// TIA Portal V16 export
// export: Created 2024-04-15T10:45:14.7081519Z, ExportSetting WithDefaults, DisplayName Totally Integrated Automation Portal, DisplayVersion V16 Update 6, DisplayName TIA Portal Version Control Interface, DisplayVersion V16 Update 2, DisplayName TIA Portal Openness, DisplayVersion V16 Update 6, DisplayName TIA Portal Test Suite Advanced, DisplayVersion V16, DisplayName SINAMICS Startdrive Advanced, DisplayVersion V16 Update 5, DisplayName SINAMICS Startdrive G130, G150, S120, S150, SINAMICS MV, S210, DisplayVersion V16 Update 5, DisplayName SINAMICS Startdrive G110M, G120, G120C, G120D, G120P, G115D, DisplayVersion V16 Update 5, DisplayName STEP 7 Professional, DisplayVersion V16 Update 6, DisplayName STEP 7 Safety, DisplayVersion V16, DisplayName WinCC Advanced, DisplayVersion V16 Update 6
FUNCTION_BLOCK "RH_OUT_2140TR"   // FB73, LAD
TITLE = Conveyor 865TR2140 outputs / Kuljetinpohja
{ S7_Optimized_Access := 'TRUE' }
AUTHOR : JLA
VERSION : 0.1
// stored: AutoNumber true, IsIECCheckEnabled false, IsRetainMemResEnabled false, MemoryReserve 100, SetENOAutomatically false, UDAEnableTagReadback false
   VAR
      Diag : "RMP_UDT_DIAG";   // Device diagnostics / Laitteen diagnostiikka
      Status : "RMP_UDT_DEV_STATUS";   // Device status information / Laitteen tilatieto
      HMI_Status : "RMP_HMI_DEV_STATUS";   // Device status information for HMI
      IO : Struct   // Device inputs and outputs / Laitteen tulot ja lähdöt
         Input : Struct
            Safety_switch : Bool;   // Safety switch / Kuljettimen turvakytkin
            Entry_pec : Bool;   // Entry photocell / Tulovalokenno
            Exit_pec : Bool;   // Exit photocell / Poistovalokenno
            Pulse_A : Bool;   // Pulse A / Rulla viivakoodin lukukohdassa
            Pulse_B : Bool;   // Pulse B
            Next_entry_pec : Bool;   // Next entry photocell / Seuraavan kuljettimen tulokenno
            Prev_exit_pec : Bool;   // Previous exit photocell / Edellisen kuljettimen poistokenno
            Man_cnv_fwd : Bool;   // Conveyor manual forward switch
            Man_cnv_rev : Bool;   // Conveyor manual reverse switch
            In_10 : Bool;
            In_11 : Bool;
            In_12 : Bool;
            In_13 : Bool;
            In_14 : Bool;
            In_15 : Bool;
            In_16 : Bool;
            In_17 : Bool;
            In_18 : Bool;
            In_19 : Bool;
            In_20 : Bool;
            In_21 : Bool;
            In_22 : Bool;
            In_23 : Bool;
            In_24 : Bool;
            In_25 : Bool;
            In_26 : Bool;
            In_27 : Bool;
            In_28 : Bool;
            In_29 : Bool;
            In_30 : Bool;
            In_31 : Bool;
            In_32 : Bool;
         END_STRUCT;
         Output : Struct
            Out_1 : Bool;
            Out_2 : Bool;
            Out_3 : Bool;
            Out_4 : Bool;
            Out_5 : Bool;
            Out_6 : Bool;
            Out_7 : Bool;
            Out_8 : Bool;
            Out_9 : Bool;
            Out_10 : Bool;
            Out_11 : Bool;
            Out_12 : Bool;
            Out_13 : Bool;
            Out_14 : Bool;
            Out_15 : Bool;
            Out_16 : Bool;
            Out_17 : Bool;
            Out_18 : Bool;
            Out_19 : Bool;
            Out_20 : Bool;
            Out_21 : Bool;
            Out_22 : Bool;
            Out_23 : Bool;
            Out_24 : Bool;
            Out_25 : Bool;
            Out_26 : Bool;
            Out_27 : Bool;
            Out_28 : Bool;
            Out_29 : Bool;
            Out_30 : Bool;
            Out_31 : Bool;
            Out_32 : Bool;
         END_STRUCT;
      END_STRUCT;
      Flags : Struct   // Device auxilary flags / Laitteen apubitit
         Speed_1 : Bool;   // Speed selection 1 / Nopeusvalinta 1
         Speed_2 : Bool;   // Speed selection 2 / Nopeusvalinta 2
         Speed_3 : Bool;   // Speed selection 3 / Nopeusvalinta 3
         Speed_4 : Bool;   // Speed selection 4 / Nopeusvalinta 4
         Data_ok : Bool;   // Roll data present / Rulladata löytyy
         Entry_pec_fault : Bool;   // Entry pec fault bit
         Exit_pec_fault : Bool;   // Exit pec fault bit
         Auto_help : Bool;   // Auto status help bit
         Buffering : Bool;   // Buffering rolls on conveyor
         Separate : Bool;   // Separating rolls at conveyor exit joint
         Separate_p : Bool;   // Separating rolls at conveyor exit joint pulse
         Stopped : Bool;   // Device stopped
         Status_Auto : Bool;
         Status_Manual : Bool;
         Sensing_Stop_manual : Bool;
         SensingStop_help : Bool;
         Sensing_Stop : Bool;
         Bit_17 : Bool;
         Bit_18 : Bool;
         Bit_19 : Bool;
         Bit_20 : Bool;
         Bit_21 : Bool;
         Bit_22 : Bool;
         Bit_23 : Bool;
         Bit_24 : Bool;
         Bit_25 : Bool;
         Bit_26 : Bool;
         Bit_27 : Bool;
         Bit_28 : Bool;
         Bit_29 : Bool;
         Bit_30 : Bool;
         Bit_31 : Bool;
         Bit_32 : Bool;
         Bit_33 : Bool;
         Bit_34 : Bool;
         Bit_35 : Bool;
         Bit_36 : Bool;
         Bit_37 : Bool;
         Bit_38 : Bool;
         Bit_39 : Bool;
         Bit_40 : Bool;
         Bit_41 : Bool;
         Bit_42 : Bool;
         Bit_43 : Bool;
         Bit_44 : Bool;
         Bit_45 : Bool;
         Bit_46 : Bool;
         Bit_47 : Bool;
         Bit_48 : Bool;
         Bit_49 : Bool;
         Bit_50 : Bool;
         Bit_51 : Bool;
         Bit_52 : Bool;
         Bit_53 : Bool;
         Bit_54 : Bool;
         Bit_55 : Bool;
         Bit_56 : Bool;
         Bit_57 : Bool;
         Bit_58 : Bool;
         Bit_59 : Bool;
         Bit_60 : Bool;
         Bit_61 : Bool;
         Bit_62 : Bool;
         Bit_63 : Bool;
      END_STRUCT;
      Data : Struct   // Device data / Laitteen data
         Data_int_1 : Int;
         Data_int_2 : Int;
         Data_int_3 : Int;
         Data_int_4 : Int;
         Data_int_5 : Int;
         Data_int_6 : Int;
         Data_int_7 : Int;
         Data_int_8 : Int;
         Data_int_9 : Int;
         Data_int_10 : Int;
         Data_int_11 : Int;
         Data_int_12 : Int;
         Data_int_13 : Int;
         Data_int_14 : Int;
         Data_int_15 : Int;
         Data_int_16 : Int;
         Data_int_17 : Int;
         Data_int_18 : Int;
         Data_int_19 : Int;
         Data_int_20 : Int;
         Data_Dint_1 : DInt;
         Data_Dint_2 : DInt;
         Data_Dint_3 : DInt;
         Data_Dint_4 : DInt;
         Data_Dint_5 : DInt;
         Data_Dint_6 : DInt;
         Data_Dint_7 : DInt;
         Data_Dint_8 : DInt;
         Data_Dint_9 : DInt;
         Data_Dint_10 : DInt;
         Data_Dint_11 : DInt;
         Data_Dint_12 : DInt;
         Data_Dint_13 : DInt;
         Data_Dint_14 : DInt;
         Data_Dint_15 : DInt;
         Data_Dint_16 : DInt;
         Data_from_prev : DWord;   // Data from previous conveyor
         Data_from_next : DWord;   // Data from next conveyor
         Data_next : DWord;   // Conveyor data for next conveyor / Kuljettimen data seuraavalle kuljettimelle
         Data_prev : DWord;   // Conveyor data for previous conveyor / Kuljettimen data edelliselle kuljettimelle
      END_STRUCT;
      Interlock : "RMP_UDT_INTERLOCK";   // Conveyor / Laitelukitukset
      Control : "RMP_UDT_CONTROL";   // Laitteen ohjaus / Device control
      Frq : "RMP_BIF_FRQ_SPD";   // Device frequency converter control / Laitteen taajuusmuuttajan ohjaus
      Drive : "RMP_FRQ_SPD";   // Device frequency converter instance
      Encoder : "RMP_BIF_CNV_ENC";   // Device encoder
      Entry_gap : "RMP_BIF_GAP_CONTROL";   // Entry gap control
      Program_Alarm : Array[1..16] of Program_Alarm;   // Device alarms
      Program_Event : Array[1..8] of Program_Alarm;   // Device events / Laitteen tapahtumat
      Device_name : String[40] := 'Slat conveyor - 865TR2140';   // Device name
      RMP_CNV_ENC_Instance : "RMP_CNV_ENC";
      RMP_CONV_DATA_Instance : "RMP_CONV_DATA";
      RMP_SERV_COUNTER_Instance : "RMP_SERV_COUNTER";
      RMP_GAP_CONTROL_Instance : "RMP_GAP_CONTROL";
      RMP_EMPTY_CNT_Instance : "RMP_EMPTY_CNT";
      RMP_PEC_FAULT_Instance_1 : "RMP_PEC_FAULT";
      RMP_PEC_FAULT_Instance_2 : "RMP_PEC_FAULT";
      Event_1_delay : TON_TIME;
      Encoder_delay : TON_TIME;
      ORG : Struct
         Start_End_Print : Bool;
         ORG_2 : Bool;
         Start_Belly_Print : Bool;
         ORG_4 : Bool;
         ORG_5 : Bool;
         ORG_6 : Bool;
         ORG_7 : Bool;
         ORG_8 : Bool;
      END_STRUCT;
      MSG_Timeout { S7_SetPoint := 'True'} : TON_TIME;
   END_VAR
   VAR_TEMP
      Temp_R : Real;
      Temp_I : Int;
      Temp_DI : DInt;
      Error : Bool;
      Replace : Struct
         Prev_rev : Bool;
         Next_fwd : Bool;
         Conveyor_data : Array[1..10] of DWord;
         Roll_width : Int;
      END_STRUCT;
      Error_nbr : Int;
   END_VAR
   // // Interlock.Fwd : eteenpäin / forward interlocks
   // // Interlock.Fwd[1] : Safety switch open / Turvakytkin auki
   // // Interlock.Fwd[2] : Exit pec on and next is not running / Poistokenno vaikuttuneena ja seuraava ei aja
   // // Interlock.Fwd[3] : Exit pec on and next is not ready
   // // Interlock.Fwd[4] : Rollers is not at down position
   // // Interlock.Fwd[5] : Entry Pec and Belly marker not in up position
   // // Interlock.Fwd[6] : Entry Pec and inkjet Marker not in up position
   // // Interlock.Fwd[7] : Area Free 2 and inkjet Marker not in up position
   // // Interlock.Fwd[8] : Roll at joint and prev is not running
   // // Interlock.Rev : taaksepäin / reverse interlocks
   // // Interlock.Rev[1] : Safety switch open / Turvakytkin auki
   // // Interlock.Rev[2] : Entry pec on and prev is not running / Tulokenno vaikuttuneena ja edeltävä ei aja
   // // Interlock.Rev[3] : Rollers is not at down position
   // // Interlock.Rev[4] : inkjet Marker 2150 not in up position
   // // Interlock.Rev[5] : Belly marker not in up position
   // // Interlock.Rev[6] : Area free 2 and inkjet Marker 2130 not in up position
   VAR_TEMP   // added for the SCL form of the ladder/FBD networks
      _w1 : Bool;
   END_VAR
BEGIN

REGION Network 1: Control area interface / Ohjausalueen rajapinta
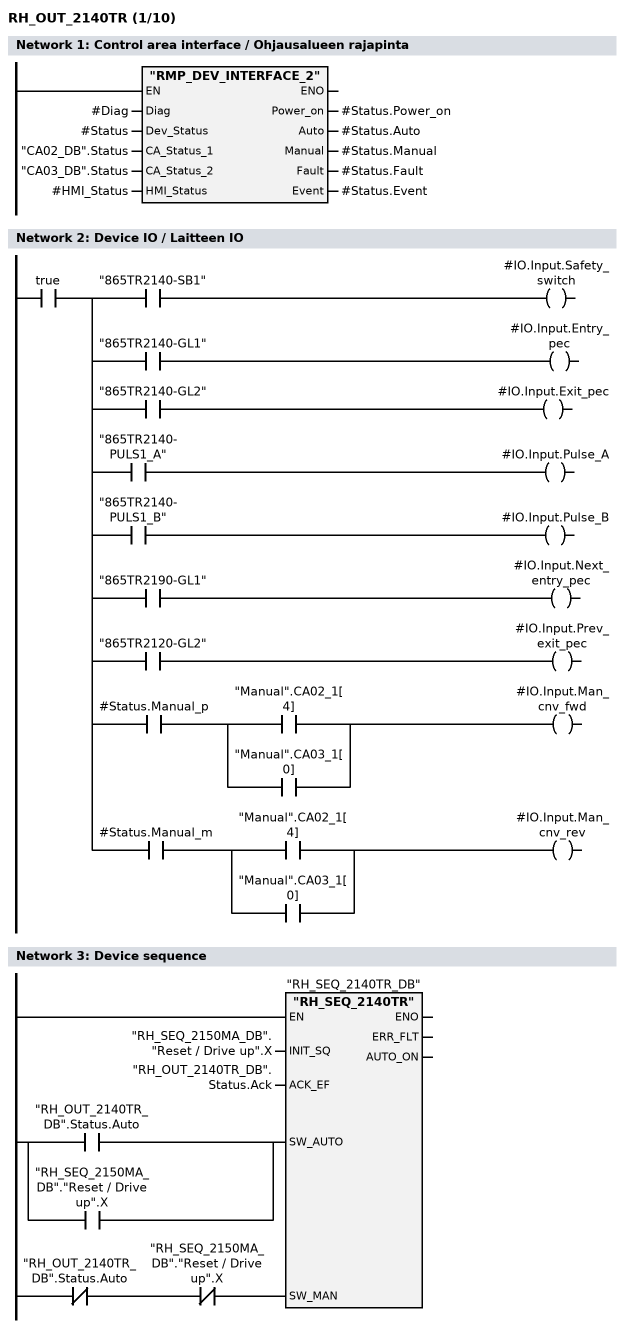
   RUNG wire#powerrail
      "RMP_DEV_INTERFACE_2"(Diag := #Diag, Dev_Status := #Status, CA_Status_1 := "CA02_DB".Status, CA_Status_2 := "CA03_DB".Status, HMI_Status := #HMI_Status, Power_on => #Status.Power_on, Auto => #Status.Auto, Manual => #Status.Manual, Fault => #Status.Fault, Event => #Status.Event)
   END_RUNG
   // the same network as SCL:
   "RMP_DEV_INTERFACE_2"(Diag := #Diag,
                         Dev_Status := #Status,
                         CA_Status_1 := "CA02_DB".Status,
                         CA_Status_2 := "CA03_DB".Status,
                         HMI_Status := #HMI_Status,
                         Power_on => #Status.Power_on,
                         Auto => #Status.Auto,
                         Manual => #Status.Manual,
                         Fault => #Status.Fault,
                         Event => #Status.Event);
END_REGION

REGION Network 2: Device IO / Laitteen IO
   RUNG wire#powerrail
      Contact( true )
      wire#w1
      Contact( "865TR2140-SB1" )
      Coil( #IO.Input.Safety_switch )
   END_RUNG
   RUNG wire#w1
      Contact( "865TR2140-GL1" )
      Coil( #IO.Input.Entry_pec )
   END_RUNG
   RUNG wire#w1
      Contact( "865TR2140-GL2" )
      Coil( #IO.Input.Exit_pec )
   END_RUNG
   RUNG wire#w1
      Contact( "865TR2140-PULS1_A" )
      Coil( #IO.Input.Pulse_A )
   END_RUNG
   RUNG wire#w1
      Contact( "865TR2140-PULS1_B" )
      Coil( #IO.Input.Pulse_B )
   END_RUNG
   RUNG wire#w1
      Contact( "865TR2190-GL1" )
      Coil( #IO.Input.Next_entry_pec )
   END_RUNG
   RUNG wire#w1
      Contact( "865TR2120-GL2" )
      Coil( #IO.Input.Prev_exit_pec )
   END_RUNG
   RUNG wire#w1
      Contact( #Status.Manual_p )
      wire#w2
      Contact( "Manual".CA02_1[4] )
      wire#w3
      Coil( #IO.Input.Man_cnv_fwd )
   END_RUNG
   RUNG wire#w2
      Contact( "Manual".CA03_1[0] )
   END_RUNG wire#w3
   RUNG wire#w1
      Contact( #Status.Manual_m )
      wire#w4
      Contact( "Manual".CA02_1[4] )
      wire#w5
      Coil( #IO.Input.Man_cnv_rev )
   END_RUNG
   RUNG wire#w4
      Contact( "Manual".CA03_1[0] )
   END_RUNG wire#w5
   // the same network as SCL:
   #IO.Input.Safety_switch := true AND "865TR2140-SB1";
   #IO.Input.Entry_pec := true AND "865TR2140-GL1";
   #IO.Input.Exit_pec := true AND "865TR2140-GL2";
   #IO.Input.Pulse_A := true AND "865TR2140-PULS1_A";
   #IO.Input.Pulse_B := true AND "865TR2140-PULS1_B";
   #IO.Input.Next_entry_pec := true AND "865TR2190-GL1";
   #IO.Input.Prev_exit_pec := true AND "865TR2120-GL2";
   #IO.Input.Man_cnv_fwd := true AND #Status.Manual_p AND ("Manual".CA02_1[4] OR "Manual".CA03_1[0]);
   #IO.Input.Man_cnv_rev := true AND #Status.Manual_m AND ("Manual".CA02_1[4] OR "Manual".CA03_1[0]);
END_REGION

REGION Network 3: Device sequence
   RUNG wire#powerrail
      "RH_SEQ_2140TR_DB"(SW_AUTO := wire#w1, SW_MAN := wire#w2, INIT_SQ := "RH_SEQ_2150MA_DB"."Reset / Drive up".X, ACK_EF := "RH_OUT_2140TR_DB".Status.Ack, ERR_FLT =>, AUTO_ON =>)
   END_RUNG
   RUNG wire#powerrail
      Contact( "RH_OUT_2140TR_DB".Status.Auto )
   END_RUNG wire#w1
   RUNG wire#powerrail
      Contact( "RH_SEQ_2150MA_DB"."Reset / Drive up".X )
   END_RUNG wire#w1
   RUNG wire#powerrail
      I_Contact( "RH_OUT_2140TR_DB".Status.Auto )
      I_Contact( "RH_SEQ_2150MA_DB"."Reset / Drive up".X )
   END_RUNG wire#w2
   // the same network as SCL:
   "RH_SEQ_2140TR_DB"(INIT_SQ := "RH_SEQ_2150MA_DB"."Reset / Drive up".X,   // "RH_SEQ_2140TR"
                      ACK_EF := "RH_OUT_2140TR_DB".Status.Ack,
                      SW_AUTO := "RH_OUT_2140TR_DB".Status.Auto OR "RH_SEQ_2150MA_DB"."Reset / Drive up".X,
                      SW_MAN := NOT "RH_OUT_2140TR_DB".Status.Auto AND NOT "RH_SEQ_2150MA_DB"."Reset / Drive up".X);
END_REGION

REGION Network 4: Device stopped information for safety door control
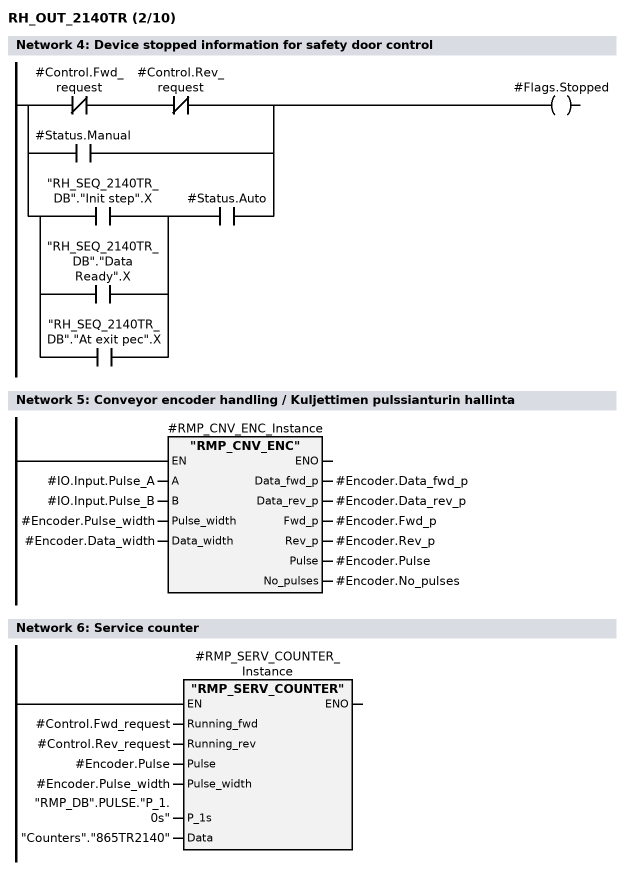
   RUNG wire#powerrail
      I_Contact( #Control.Fwd_request )
      I_Contact( #Control.Rev_request )
      wire#w1
      Coil( #Flags.Stopped )
   END_RUNG
   RUNG wire#powerrail
      Contact( #Status.Manual )
   END_RUNG wire#w1
   RUNG wire#powerrail
      Contact( "RH_SEQ_2140TR_DB"."Init step".X )
      wire#w2
      Contact( #Status.Auto )
   END_RUNG wire#w1
   RUNG wire#powerrail
      Contact( "RH_SEQ_2140TR_DB"."Data Ready".X )
   END_RUNG wire#w2
   RUNG wire#powerrail
      Contact( "RH_SEQ_2140TR_DB"."At exit pec".X )
   END_RUNG wire#w2
   // the same network as SCL:
   #Flags.Stopped := (NOT #Control.Fwd_request AND NOT #Control.Rev_request) OR #Status.Manual OR (("RH_SEQ_2140TR_DB"."Init step".X OR "RH_SEQ_2140TR_DB"."Data Ready".X OR "RH_SEQ_2140TR_DB"."At exit pec".X) AND #Status.Auto);
END_REGION

REGION Network 5: Conveyor encoder handling / Kuljettimen pulssianturin hallinta
   RUNG wire#powerrail
      #RMP_CNV_ENC_Instance("A" := #IO.Input.Pulse_A, "B" := #IO.Input.Pulse_B, Pulse_width := #Encoder.Pulse_width, Data_width := #Encoder.Data_width, Data_fwd_p => #Encoder.Data_fwd_p, Data_rev_p => #Encoder.Data_rev_p, Fwd_p => #Encoder.Fwd_p, Rev_p => #Encoder.Rev_p, Pulse => #Encoder.Pulse, No_pulses => #Encoder.No_pulses)
   END_RUNG
   // the same network as SCL:
   #RMP_CNV_ENC_Instance("A" := #IO.Input.Pulse_A,   // "RMP_CNV_ENC"
                         "B" := #IO.Input.Pulse_B,
                         Pulse_width := #Encoder.Pulse_width,
                         Data_width := #Encoder.Data_width,
                         Data_fwd_p => #Encoder.Data_fwd_p,
                         Data_rev_p => #Encoder.Data_rev_p,
                         Fwd_p => #Encoder.Fwd_p,
                         Rev_p => #Encoder.Rev_p,
                         Pulse => #Encoder.Pulse,
                         No_pulses => #Encoder.No_pulses);
END_REGION

REGION Network 6: Service counter
   RUNG wire#powerrail
      #RMP_SERV_COUNTER_Instance(Running_fwd := #Control.Fwd_request, Running_rev := #Control.Rev_request, Pulse := #Encoder.Pulse, Pulse_width := #Encoder.Pulse_width, P_1s := "RMP_DB".PULSE."P_1.0s", Data := "Counters"."865TR2140")
   END_RUNG
   // the same network as SCL:
   #RMP_SERV_COUNTER_Instance(Running_fwd := #Control.Fwd_request,   // "RMP_SERV_COUNTER"
                           Running_rev := #Control.Rev_request,
                           Pulse := #Encoder.Pulse,
                           Pulse_width := #Encoder.Pulse_width,
                           P_1s := "RMP_DB".PULSE."P_1.0s",
                           Data := "Counters"."865TR2140");
END_REGION

REGION Network 7: Conveyor forward interlock / Kuljetin eteenpäin, lukitukset
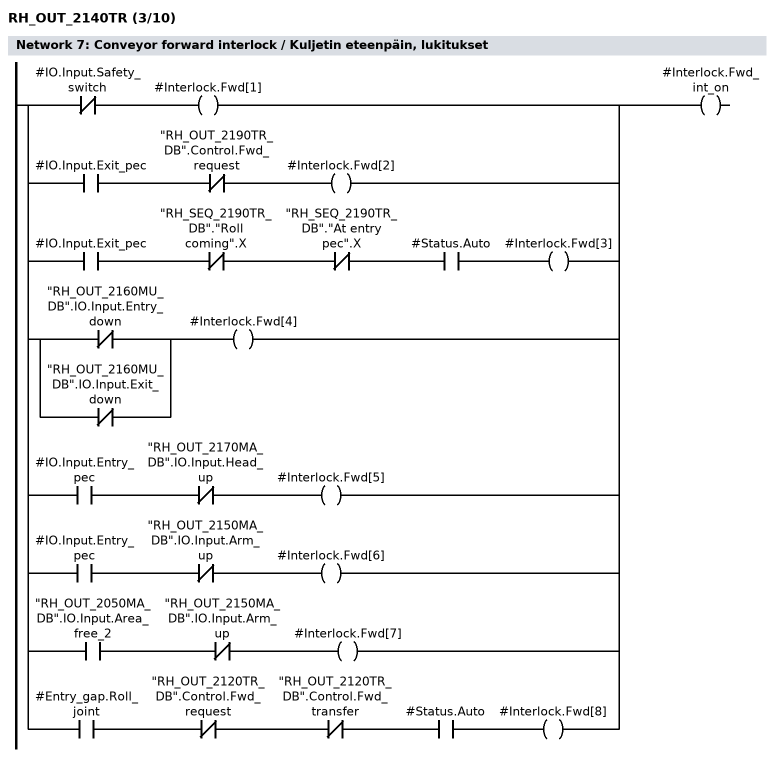
   RUNG wire#powerrail
      I_Contact( #IO.Input.Safety_switch )
      Coil( #Interlock.Fwd[1] )
      wire#w1
      Coil( #Interlock.Fwd_int_on )
   END_RUNG
   RUNG wire#powerrail
      Contact( #IO.Input.Exit_pec )
      I_Contact( "RH_OUT_2190TR_DB".Control.Fwd_request )
      Coil( #Interlock.Fwd[2] )
   END_RUNG wire#w1
   RUNG wire#powerrail
      Contact( #IO.Input.Exit_pec )
      I_Contact( "RH_SEQ_2190TR_DB"."Roll coming".X )
      I_Contact( "RH_SEQ_2190TR_DB"."At entry pec".X )
      Contact( #Status.Auto )
      Coil( #Interlock.Fwd[3] )
   END_RUNG wire#w1
   RUNG wire#powerrail
      I_Contact( "RH_OUT_2160MU_DB".IO.Input.Entry_down )
      wire#w2
      Coil( #Interlock.Fwd[4] )
   END_RUNG wire#w1
   RUNG wire#powerrail
      I_Contact( "RH_OUT_2160MU_DB".IO.Input.Exit_down )
   END_RUNG wire#w2
   RUNG wire#powerrail
      Contact( #IO.Input.Entry_pec )
      I_Contact( "RH_OUT_2170MA_DB".IO.Input.Head_up )
      Coil( #Interlock.Fwd[5] )
   END_RUNG wire#w1
   RUNG wire#powerrail
      Contact( #IO.Input.Entry_pec )
      I_Contact( "RH_OUT_2150MA_DB".IO.Input.Arm_up )
      Coil( #Interlock.Fwd[6] )
   END_RUNG wire#w1
   RUNG wire#powerrail
      Contact( "RH_OUT_2050MA_DB".IO.Input.Area_free_2 )
      I_Contact( "RH_OUT_2150MA_DB".IO.Input.Arm_up )
      Coil( #Interlock.Fwd[7] )
   END_RUNG wire#w1
   RUNG wire#powerrail
      Contact( #Entry_gap.Roll_joint )
      I_Contact( "RH_OUT_2120TR_DB".Control.Fwd_request )
      I_Contact( "RH_OUT_2120TR_DB".Control.Fwd_transfer )
      Contact( #Status.Auto )
      Coil( #Interlock.Fwd[8] )
   END_RUNG wire#w1
   // the same network as SCL:
   #Interlock.Fwd[1] := NOT #IO.Input.Safety_switch;
   #Interlock.Fwd[2] := #IO.Input.Exit_pec AND NOT "RH_OUT_2190TR_DB".Control.Fwd_request;
   #Interlock.Fwd[3] := #IO.Input.Exit_pec AND NOT "RH_SEQ_2190TR_DB"."Roll coming".X AND NOT "RH_SEQ_2190TR_DB"."At entry pec".X AND #Status.Auto;
   #Interlock.Fwd[4] := NOT "RH_OUT_2160MU_DB".IO.Input.Entry_down OR NOT "RH_OUT_2160MU_DB".IO.Input.Exit_down;
   #Interlock.Fwd[5] := #IO.Input.Entry_pec AND NOT "RH_OUT_2170MA_DB".IO.Input.Head_up;
   #Interlock.Fwd[6] := #IO.Input.Entry_pec AND NOT "RH_OUT_2150MA_DB".IO.Input.Arm_up;
   #Interlock.Fwd[7] := "RH_OUT_2050MA_DB".IO.Input.Area_free_2 AND NOT "RH_OUT_2150MA_DB".IO.Input.Arm_up;
   #Interlock.Fwd[8] := #Entry_gap.Roll_joint AND NOT "RH_OUT_2120TR_DB".Control.Fwd_request AND NOT "RH_OUT_2120TR_DB".Control.Fwd_transfer AND #Status.Auto;
   #Interlock.Fwd_int_on := NOT #IO.Input.Safety_switch OR (#IO.Input.Exit_pec AND NOT "RH_OUT_2190TR_DB".Control.Fwd_request) OR (#IO.Input.Exit_pec AND NOT "RH_SEQ_2190TR_DB"."Roll coming".X AND NOT "RH_SEQ_2190TR_DB"."At entry pec".X AND #Status.Auto) OR NOT "RH_OUT_2160MU_DB".IO.Input.Entry_down OR NOT "RH_OUT_2160MU_DB".IO.Input.Exit_down OR (#IO.Input.Entry_pec AND NOT "RH_OUT_2170MA_DB".IO.Input.Head_up) OR (#IO.Input.Entry_pec AND NOT "RH_OUT_2150MA_DB".IO.Input.Arm_up) OR ("RH_OUT_2050MA_DB".IO.Input.Area_free_2 AND NOT "RH_OUT_2150MA_DB".IO.Input.Arm_up) OR (#Entry_gap.Roll_joint AND NOT "RH_OUT_2120TR_DB".Control.Fwd_request AND NOT "RH_OUT_2120TR_DB".Control.Fwd_transfer AND #Status.Auto);
END_REGION

REGION Network 8: Conveyor forward / Kuljetin eteenpäin
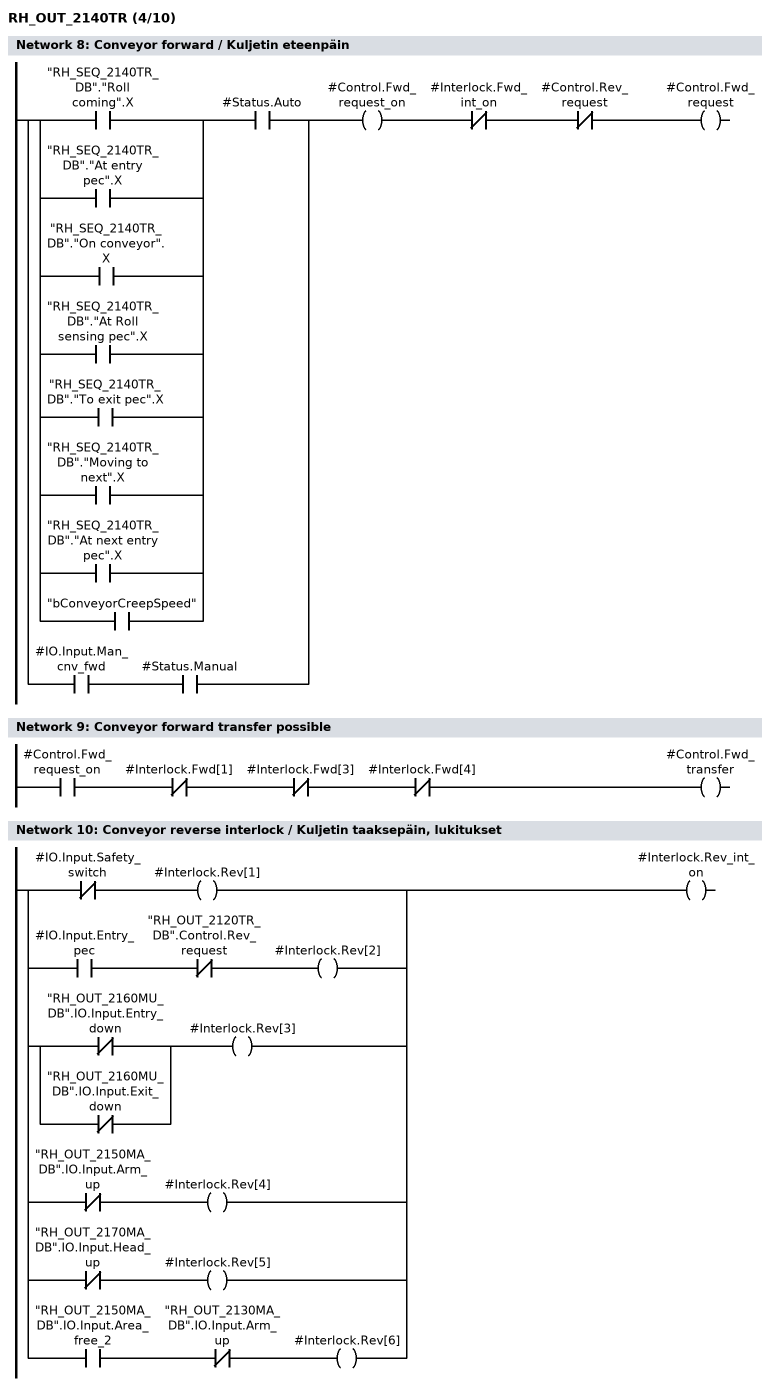
   RUNG wire#powerrail
      Contact( "RH_SEQ_2140TR_DB"."Roll coming".X )
      wire#w1
      Contact( #Status.Auto )
      wire#w2
      Coil( #Control.Fwd_request_on )
      I_Contact( #Interlock.Fwd_int_on )
      I_Contact( #Control.Rev_request )
      Coil( #Control.Fwd_request )
   END_RUNG
   RUNG wire#powerrail
      Contact( "RH_SEQ_2140TR_DB"."At entry pec".X )
   END_RUNG wire#w1
   RUNG wire#powerrail
      Contact( "RH_SEQ_2140TR_DB"."On conveyor".X )
   END_RUNG wire#w1
   RUNG wire#powerrail
      Contact( "RH_SEQ_2140TR_DB"."At Roll sensing pec".X )
   END_RUNG wire#w1
   RUNG wire#powerrail
      Contact( "RH_SEQ_2140TR_DB"."To exit pec".X )
   END_RUNG wire#w1
   RUNG wire#powerrail
      Contact( "RH_SEQ_2140TR_DB"."Moving to next".X )
   END_RUNG wire#w1
   RUNG wire#powerrail
      Contact( "RH_SEQ_2140TR_DB"."At next entry pec".X )
   END_RUNG wire#w1
   RUNG wire#powerrail
      Contact( "bConveyorCreepSpeed" )
   END_RUNG wire#w1
   RUNG wire#powerrail
      Contact( #IO.Input.Man_cnv_fwd )
      Contact( #Status.Manual )
   END_RUNG wire#w2
   // the same network as SCL:
   #Control.Fwd_request_on := (("RH_SEQ_2140TR_DB"."Roll coming".X OR "RH_SEQ_2140TR_DB"."At entry pec".X OR "RH_SEQ_2140TR_DB"."On conveyor".X OR "RH_SEQ_2140TR_DB"."At Roll sensing pec".X OR "RH_SEQ_2140TR_DB"."To exit pec".X OR "RH_SEQ_2140TR_DB"."Moving to next".X OR "RH_SEQ_2140TR_DB"."At next entry pec".X OR "bConveyorCreepSpeed") AND #Status.Auto) OR (#IO.Input.Man_cnv_fwd AND #Status.Manual);
   #Control.Fwd_request := #Control.Fwd_request_on AND NOT #Interlock.Fwd_int_on AND NOT #Control.Rev_request;
END_REGION

REGION Network 9: Conveyor forward transfer possible
   RUNG wire#powerrail
      Contact( #Control.Fwd_request_on )
      I_Contact( #Interlock.Fwd[1] )
      I_Contact( #Interlock.Fwd[3] )
      I_Contact( #Interlock.Fwd[4] )
      Coil( #Control.Fwd_transfer )
   END_RUNG
   // the same network as SCL:
   #Control.Fwd_transfer := #Control.Fwd_request_on AND NOT #Interlock.Fwd[1] AND NOT #Interlock.Fwd[3] AND NOT #Interlock.Fwd[4];
END_REGION

REGION Network 10: Conveyor reverse interlock / Kuljetin taaksepäin, lukitukset
   RUNG wire#powerrail
      I_Contact( #IO.Input.Safety_switch )
      Coil( #Interlock.Rev[1] )
      wire#w1
      Coil( #Interlock.Rev_int_on )
   END_RUNG
   RUNG wire#powerrail
      Contact( #IO.Input.Entry_pec )
      I_Contact( "RH_OUT_2120TR_DB".Control.Rev_request )
      Coil( #Interlock.Rev[2] )
   END_RUNG wire#w1
   RUNG wire#powerrail
      I_Contact( "RH_OUT_2160MU_DB".IO.Input.Entry_down )
      wire#w2
      Coil( #Interlock.Rev[3] )
   END_RUNG wire#w1
   RUNG wire#powerrail
      I_Contact( "RH_OUT_2160MU_DB".IO.Input.Exit_down )
   END_RUNG wire#w2
   RUNG wire#powerrail
      I_Contact( "RH_OUT_2150MA_DB".IO.Input.Arm_up )
      Coil( #Interlock.Rev[4] )
   END_RUNG wire#w1
   RUNG wire#powerrail
      I_Contact( "RH_OUT_2170MA_DB".IO.Input.Head_up )
      Coil( #Interlock.Rev[5] )
   END_RUNG wire#w1
   RUNG wire#powerrail
      Contact( "RH_OUT_2150MA_DB".IO.Input.Area_free_2 )
      I_Contact( "RH_OUT_2130MA_DB".IO.Input.Arm_up )
      Coil( #Interlock.Rev[6] )
   END_RUNG wire#w1
   // the same network as SCL:
   #Interlock.Rev[1] := NOT #IO.Input.Safety_switch;
   #Interlock.Rev[2] := #IO.Input.Entry_pec AND NOT "RH_OUT_2120TR_DB".Control.Rev_request;
   #Interlock.Rev[3] := NOT "RH_OUT_2160MU_DB".IO.Input.Entry_down OR NOT "RH_OUT_2160MU_DB".IO.Input.Exit_down;
   #Interlock.Rev[4] := NOT "RH_OUT_2150MA_DB".IO.Input.Arm_up;
   #Interlock.Rev[5] := NOT "RH_OUT_2170MA_DB".IO.Input.Head_up;
   #Interlock.Rev[6] := "RH_OUT_2150MA_DB".IO.Input.Area_free_2 AND NOT "RH_OUT_2130MA_DB".IO.Input.Arm_up;
   #Interlock.Rev_int_on := NOT #IO.Input.Safety_switch OR (#IO.Input.Entry_pec AND NOT "RH_OUT_2120TR_DB".Control.Rev_request) OR NOT "RH_OUT_2160MU_DB".IO.Input.Entry_down OR NOT "RH_OUT_2160MU_DB".IO.Input.Exit_down OR NOT "RH_OUT_2150MA_DB".IO.Input.Arm_up OR NOT "RH_OUT_2170MA_DB".IO.Input.Head_up OR ("RH_OUT_2150MA_DB".IO.Input.Area_free_2 AND NOT "RH_OUT_2130MA_DB".IO.Input.Arm_up);
END_REGION

REGION Network 11: Conveyor reverse / Kuljetin taaksepäin
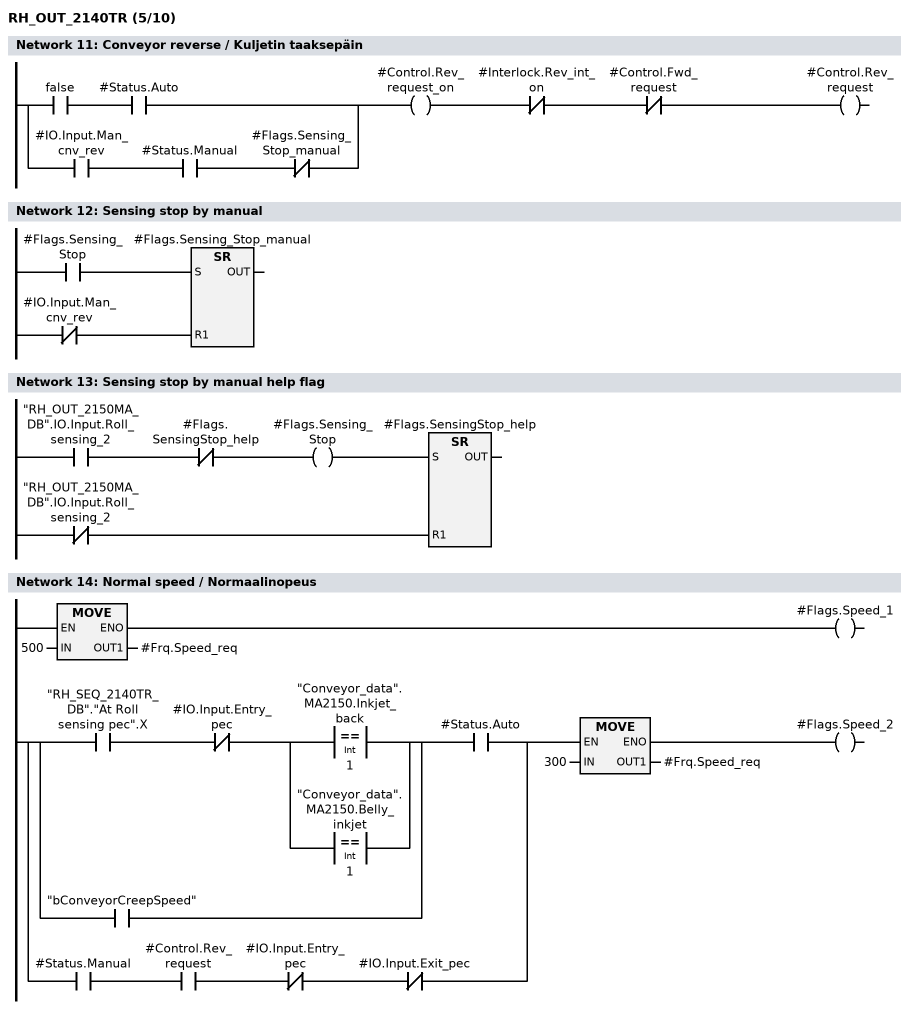
   RUNG wire#powerrail
      Contact( false )
      Contact( #Status.Auto )
      wire#w1
      Coil( #Control.Rev_request_on )
      I_Contact( #Interlock.Rev_int_on )
      I_Contact( #Control.Fwd_request )
      Coil( #Control.Rev_request )
   END_RUNG
   RUNG wire#powerrail
      Contact( #IO.Input.Man_cnv_rev )
      Contact( #Status.Manual )
      I_Contact( #Flags.Sensing_Stop_manual )
   END_RUNG wire#w1
   // the same network as SCL:
   #Control.Rev_request_on := (false AND #Status.Auto) OR (#IO.Input.Man_cnv_rev AND #Status.Manual AND NOT #Flags.Sensing_Stop_manual);
   #Control.Rev_request := #Control.Rev_request_on AND NOT #Interlock.Rev_int_on AND NOT #Control.Fwd_request;
END_REGION

REGION Network 12: Sensing stop by manual
   RUNG wire#powerrail
      Contact( #Flags.Sensing_Stop )
      S_SR(operand := #Flags.Sensing_Stop_manual, r1 := wire#w1)
   END_RUNG
   RUNG wire#powerrail
      I_Contact( #IO.Input.Man_cnv_rev )
   END_RUNG wire#w1
   // the same network as SCL:
   IF #Flags.Sensing_Stop THEN
       #Flags.Sensing_Stop_manual := TRUE;   // SR flip-flop
   END_IF;
   IF NOT #IO.Input.Man_cnv_rev THEN #Flags.Sensing_Stop_manual := FALSE; END_IF;
END_REGION

REGION Network 13: Sensing stop by manual help flag
   RUNG wire#powerrail
      Contact( "RH_OUT_2150MA_DB".IO.Input.Roll_sensing_2 )
      I_Contact( #Flags.SensingStop_help )
      Coil( #Flags.Sensing_Stop )
      S_SR(operand := #Flags.SensingStop_help, r1 := wire#w1)
   END_RUNG
   RUNG wire#powerrail
      I_Contact( "RH_OUT_2150MA_DB".IO.Input.Roll_sensing_2 )
   END_RUNG wire#w1
   // the same network as SCL:
   #Flags.Sensing_Stop := "RH_OUT_2150MA_DB".IO.Input.Roll_sensing_2 AND NOT #Flags.SensingStop_help;
   IF #Flags.Sensing_Stop THEN
       #Flags.SensingStop_help := TRUE;   // SR flip-flop
   END_IF;
   IF NOT "RH_OUT_2150MA_DB".IO.Input.Roll_sensing_2 THEN #Flags.SensingStop_help := FALSE; END_IF;
END_REGION

REGION Network 14: Normal speed / Normaalinopeus
   RUNG wire#powerrail
      { S7_GenerateENO := "TRUE" } Move(in := 500, out1 => #Frq.Speed_req)
      Coil( #Flags.Speed_1 )
   END_RUNG
   RUNG wire#powerrail
      Contact( "RH_SEQ_2140TR_DB"."At Roll sensing pec".X )
      I_Contact( #IO.Input.Entry_pec )
      wire#w1
      { S7_Templates := "SrcType := Int" } EQ_Contact(in1 := "Conveyor_data".MA2150.Inkjet_back, in2 := 1)
      wire#w2
      Contact( #Status.Auto )
      wire#w3
      { S7_GenerateENO := "TRUE" } Move(in := 300, out1 => #Frq.Speed_req)
      Coil( #Flags.Speed_2 )
   END_RUNG
   RUNG wire#w1
      { S7_Templates := "SrcType := Int" } EQ_Contact(in1 := "Conveyor_data".MA2150.Belly_inkjet, in2 := 1)
   END_RUNG wire#w2
   RUNG wire#powerrail
      Contact( "bConveyorCreepSpeed" )
   END_RUNG wire#w2
   RUNG wire#powerrail
      Contact( #Status.Manual )
      Contact( #Control.Rev_request )
      I_Contact( #IO.Input.Entry_pec )
      I_Contact( #IO.Input.Exit_pec )
   END_RUNG wire#w3
   // the same network as SCL:
   // ENO of a box is taken as its EN; it also drops when the box reports an error
   #Frq.Speed_req := 500;
   #Flags.Speed_1 := TRUE;
   #_w1 := ((("RH_SEQ_2140TR_DB"."At Roll sensing pec".X AND NOT #IO.Input.Entry_pec AND (("Conveyor_data".MA2150.Inkjet_back = 1) OR ("Conveyor_data".MA2150.Belly_inkjet = 1))) OR "bConveyorCreepSpeed") AND #Status.Auto) OR (#Status.Manual AND #Control.Rev_request AND NOT #IO.Input.Entry_pec AND NOT #IO.Input.Exit_pec);
   IF #_w1 THEN #Frq.Speed_req := 300; END_IF;
   #Flags.Speed_2 := #_w1;
END_REGION

REGION Network 15: Fast speed on roll transfers
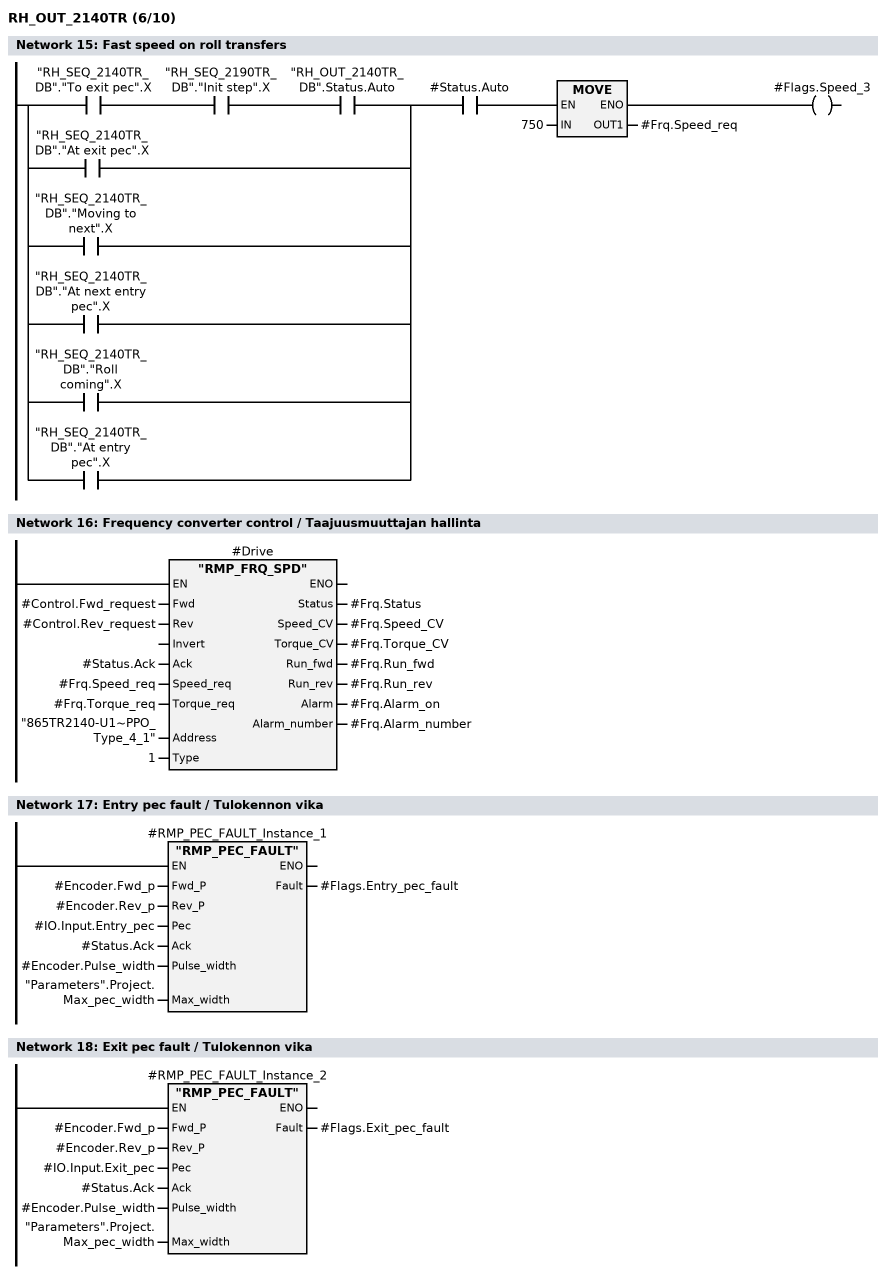
   RUNG wire#powerrail
      Contact( "RH_SEQ_2140TR_DB"."To exit pec".X )
      Contact( "RH_SEQ_2190TR_DB"."Init step".X )
      Contact( "RH_OUT_2140TR_DB".Status.Auto )
      wire#w1
      Contact( #Status.Auto )
      { S7_GenerateENO := "TRUE" } Move(in := 750, out1 => #Frq.Speed_req)
      Coil( #Flags.Speed_3 )
   END_RUNG
   RUNG wire#powerrail
      Contact( "RH_SEQ_2140TR_DB"."At exit pec".X )
   END_RUNG wire#w1
   RUNG wire#powerrail
      Contact( "RH_SEQ_2140TR_DB"."Moving to next".X )
   END_RUNG wire#w1
   RUNG wire#powerrail
      Contact( "RH_SEQ_2140TR_DB"."At next entry pec".X )
   END_RUNG wire#w1
   RUNG wire#powerrail
      Contact( "RH_SEQ_2140TR_DB"."Roll coming".X )
   END_RUNG wire#w1
   RUNG wire#powerrail
      Contact( "RH_SEQ_2140TR_DB"."At entry pec".X )
   END_RUNG wire#w1
   // the same network as SCL:
   // ENO of a box is taken as its EN; it also drops when the box reports an error
   #_w1 := (("RH_SEQ_2140TR_DB"."To exit pec".X AND "RH_SEQ_2190TR_DB"."Init step".X AND "RH_OUT_2140TR_DB".Status.Auto) OR "RH_SEQ_2140TR_DB"."At exit pec".X OR "RH_SEQ_2140TR_DB"."Moving to next".X OR "RH_SEQ_2140TR_DB"."At next entry pec".X OR "RH_SEQ_2140TR_DB"."Roll coming".X OR "RH_SEQ_2140TR_DB"."At entry pec".X) AND #Status.Auto;
   IF #_w1 THEN #Frq.Speed_req := 750; END_IF;
   #Flags.Speed_3 := #_w1;
END_REGION

REGION Network 16: Frequency converter control / Taajuusmuuttajan hallinta
   RUNG wire#powerrail
      #Drive(Fwd := #Control.Fwd_request, Rev := #Control.Rev_request, Invert :=, Ack := #Status.Ack, Speed_req := #Frq.Speed_req, Torque_req := #Frq.Torque_req, Address := "865TR2140-U1~PPO_Type_4_1", "Type" := 1, Status => #Frq.Status, Speed_CV => #Frq.Speed_CV, Torque_CV => #Frq.Torque_CV, Run_fwd => #Frq.Run_fwd, Run_rev => #Frq.Run_rev, Alarm => #Frq.Alarm_on, Alarm_number => #Frq.Alarm_number)
   END_RUNG
   // the same network as SCL:
   #Drive(Fwd := #Control.Fwd_request,   // "RMP_FRQ_SPD"
          Rev := #Control.Rev_request,
          Ack := #Status.Ack,
          Speed_req := #Frq.Speed_req,
          Torque_req := #Frq.Torque_req,
          Address := "865TR2140-U1~PPO_Type_4_1",
          "Type" := 1,
          Status => #Frq.Status,
          Speed_CV => #Frq.Speed_CV,
          Torque_CV => #Frq.Torque_CV,
          Run_fwd => #Frq.Run_fwd,
          Run_rev => #Frq.Run_rev,
          Alarm => #Frq.Alarm_on,
          Alarm_number => #Frq.Alarm_number);
END_REGION

REGION Network 17: Entry pec fault / Tulokennon vika
   RUNG wire#powerrail
      #RMP_PEC_FAULT_Instance_1(Fwd_P := #Encoder.Fwd_p, Rev_P := #Encoder.Rev_p, Pec := #IO.Input.Entry_pec, Ack := #Status.Ack, Pulse_width := #Encoder.Pulse_width, Max_width := "Parameters".Project.Max_pec_width, Fault => #Flags.Entry_pec_fault)
   END_RUNG
   // the same network as SCL:
   #RMP_PEC_FAULT_Instance_1(Fwd_P := #Encoder.Fwd_p,   // "RMP_PEC_FAULT"
                           Rev_P := #Encoder.Rev_p,
                           Pec := #IO.Input.Entry_pec,
                           Ack := #Status.Ack,
                           Pulse_width := #Encoder.Pulse_width,
                           Max_width := "Parameters".Project.Max_pec_width,
                           Fault => #Flags.Entry_pec_fault);
END_REGION

REGION Network 18: Exit pec fault / Tulokennon vika
   RUNG wire#powerrail
      #RMP_PEC_FAULT_Instance_2(Fwd_P := #Encoder.Fwd_p, Rev_P := #Encoder.Rev_p, Pec := #IO.Input.Exit_pec, Ack := #Status.Ack, Pulse_width := #Encoder.Pulse_width, Max_width := "Parameters".Project.Max_pec_width, Fault => #Flags.Exit_pec_fault)
   END_RUNG
   // the same network as SCL:
   #RMP_PEC_FAULT_Instance_2(Fwd_P := #Encoder.Fwd_p,   // "RMP_PEC_FAULT"
                           Rev_P := #Encoder.Rev_p,
                           Pec := #IO.Input.Exit_pec,
                           Ack := #Status.Ack,
                           Pulse_width := #Encoder.Pulse_width,
                           Max_width := "Parameters".Project.Max_pec_width,
                           Fault => #Flags.Exit_pec_fault);
END_REGION

REGION Network 19: Roll coming to conveyor from entry side
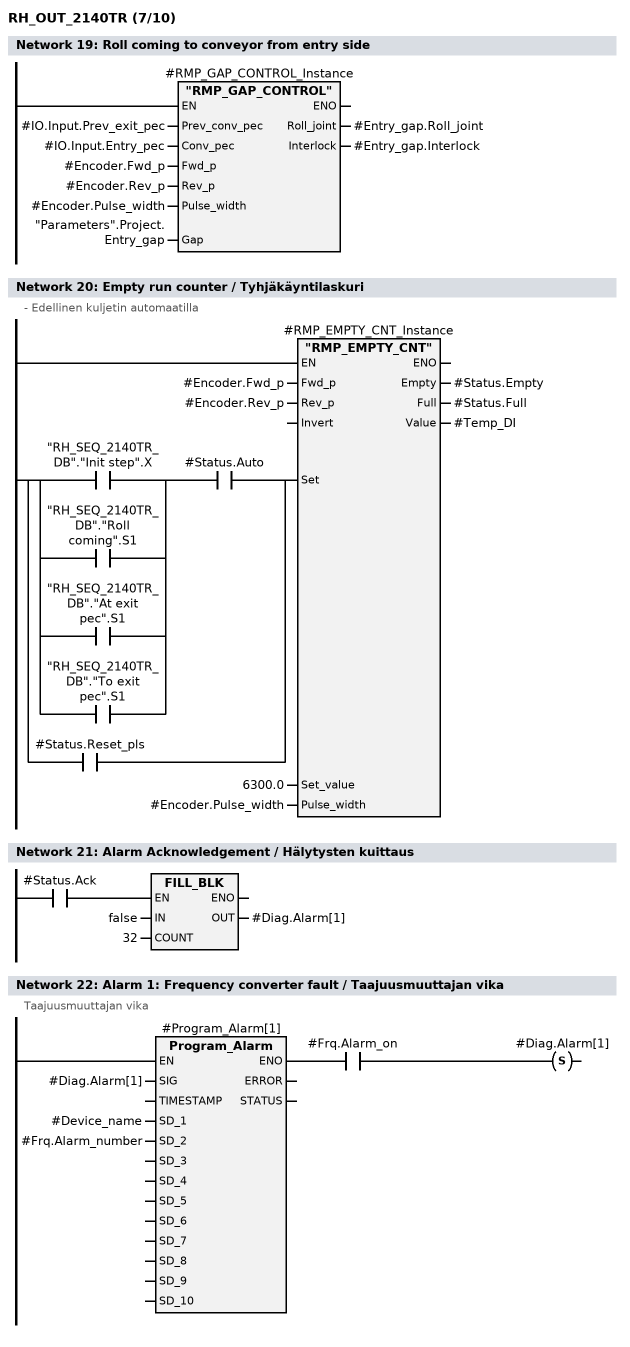
   RUNG wire#powerrail
      #RMP_GAP_CONTROL_Instance(Prev_conv_pec := #IO.Input.Prev_exit_pec, Conv_pec := #IO.Input.Entry_pec, Fwd_p := #Encoder.Fwd_p, Rev_p := #Encoder.Rev_p, Pulse_width := #Encoder.Pulse_width, Gap := "Parameters".Project.Entry_gap, Roll_joint => #Entry_gap.Roll_joint, Interlock => #Entry_gap.Interlock)
   END_RUNG
   // the same network as SCL:
   #RMP_GAP_CONTROL_Instance(Prev_conv_pec := #IO.Input.Prev_exit_pec,   // "RMP_GAP_CONTROL"
                           Conv_pec := #IO.Input.Entry_pec,
                           Fwd_p := #Encoder.Fwd_p,
                           Rev_p := #Encoder.Rev_p,
                           Pulse_width := #Encoder.Pulse_width,
                           Gap := "Parameters".Project.Entry_gap,
                           Roll_joint => #Entry_gap.Roll_joint,
                           Interlock => #Entry_gap.Interlock);
END_REGION

REGION Network 20: Empty run counter / Tyhjäkäyntilaskuri
   // - Edellinen kuljetin automaatilla
   RUNG wire#powerrail
      #RMP_EMPTY_CNT_Instance(Set := wire#w2, Fwd_p := #Encoder.Fwd_p, Rev_p := #Encoder.Rev_p, Invert :=, Set_value := 6300.0, Pulse_width := #Encoder.Pulse_width, Empty => #Status.Empty, Full => #Status.Full, Value => #Temp_DI)
   END_RUNG
   RUNG wire#powerrail
      Contact( "RH_SEQ_2140TR_DB"."Init step".X )
      wire#w1
      Contact( #Status.Auto )
   END_RUNG wire#w2
   RUNG wire#powerrail
      Contact( "RH_SEQ_2140TR_DB"."Roll coming".S1 )
   END_RUNG wire#w1
   RUNG wire#powerrail
      Contact( "RH_SEQ_2140TR_DB"."At exit pec".S1 )
   END_RUNG wire#w1
   RUNG wire#powerrail
      Contact( "RH_SEQ_2140TR_DB"."To exit pec".S1 )
   END_RUNG wire#w1
   RUNG wire#powerrail
      Contact( #Status.Reset_pls )
   END_RUNG wire#w2
   // the same network as SCL:
   #RMP_EMPTY_CNT_Instance(Fwd_p := #Encoder.Fwd_p,   // "RMP_EMPTY_CNT"
                           Rev_p := #Encoder.Rev_p,
                           Set := (("RH_SEQ_2140TR_DB"."Init step".X OR "RH_SEQ_2140TR_DB"."Roll coming".S1 OR "RH_SEQ_2140TR_DB"."At exit pec".S1 OR "RH_SEQ_2140TR_DB"."To exit pec".S1) AND #Status.Auto) OR #Status.Reset_pls,
                           Set_value := 6300.0,
                           Pulse_width := #Encoder.Pulse_width,
                           Empty => #Status.Empty,
                           Full => #Status.Full,
                           Value => #Temp_DI);
END_REGION

REGION Network 21: Alarm Acknowledgement / Hälytysten kuittaus
   RUNG wire#powerrail
      Contact( #Status.Ack )
      FillBlockI(in := false, count := 32, out => #Diag.Alarm[1])
   END_RUNG
   // the same network as SCL:
   IF #Status.Ack THEN FILL_BLK(IN := false, COUNT := 32, OUT => #Diag.Alarm[1]); END_IF;
END_REGION

REGION Network 22: Alarm 1: Frequency converter fault / Taajuusmuuttajan vika
   // Taajuusmuuttajan vika
   RUNG wire#powerrail
      #Program_Alarm[1].Program_Alarm(SIG := #Diag.Alarm[1], TIMESTAMP :=, SD_1 := #Device_name, SD_2 := #Frq.Alarm_number, SD_3 :=, SD_4 :=, SD_5 :=, SD_6 :=, SD_7 :=, SD_8 :=, SD_9 :=, SD_10 :=, Error =>, Status =>)
      Contact( #Frq.Alarm_on )
      S_Coil( #Diag.Alarm[1] )
   END_RUNG
   // the same network as SCL:
   #Program_Alarm[1](SIG := #Diag.Alarm[1], SD_1 := #Device_name, SD_2 := #Frq.Alarm_number, ENO => #_w1);   // Program_Alarm
   IF #_w1 AND #Frq.Alarm_on THEN #Diag.Alarm[1] := TRUE; END_IF;
END_REGION

REGION Network 23: Alarm 2: Safety switch open / Turvakytkin auki
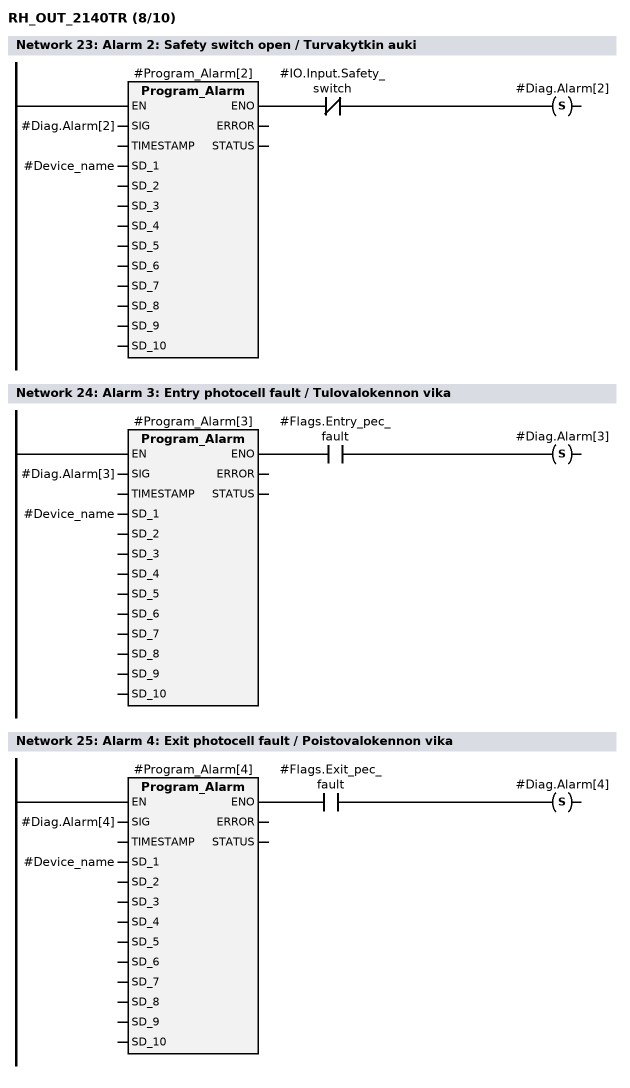
   RUNG wire#powerrail
      #Program_Alarm[2].Program_Alarm(SIG := #Diag.Alarm[2], TIMESTAMP :=, SD_1 := #Device_name, SD_2 :=, SD_3 :=, SD_4 :=, SD_5 :=, SD_6 :=, SD_7 :=, SD_8 :=, SD_9 :=, SD_10 :=, Error =>, Status =>)
      I_Contact( #IO.Input.Safety_switch )
      S_Coil( #Diag.Alarm[2] )
   END_RUNG
   // the same network as SCL:
   #Program_Alarm[2](SIG := #Diag.Alarm[2], SD_1 := #Device_name, ENO => #_w1);   // Program_Alarm
   IF #_w1 AND NOT #IO.Input.Safety_switch THEN #Diag.Alarm[2] := TRUE; END_IF;
END_REGION

REGION Network 24: Alarm 3: Entry photocell fault / Tulovalokennon vika
   RUNG wire#powerrail
      #Program_Alarm[3].Program_Alarm(SIG := #Diag.Alarm[3], TIMESTAMP :=, SD_1 := #Device_name, SD_2 :=, SD_3 :=, SD_4 :=, SD_5 :=, SD_6 :=, SD_7 :=, SD_8 :=, SD_9 :=, SD_10 :=, Error =>, Status =>)
      Contact( #Flags.Entry_pec_fault )
      S_Coil( #Diag.Alarm[3] )
   END_RUNG
   // the same network as SCL:
   #Program_Alarm[3](SIG := #Diag.Alarm[3], SD_1 := #Device_name, ENO => #_w1);   // Program_Alarm
   IF #_w1 AND #Flags.Entry_pec_fault THEN #Diag.Alarm[3] := TRUE; END_IF;
END_REGION

REGION Network 25: Alarm 4: Exit photocell fault / Poistovalokennon vika
   RUNG wire#powerrail
      #Program_Alarm[4].Program_Alarm(SIG := #Diag.Alarm[4], TIMESTAMP :=, SD_1 := #Device_name, SD_2 :=, SD_3 :=, SD_4 :=, SD_5 :=, SD_6 :=, SD_7 :=, SD_8 :=, SD_9 :=, SD_10 :=, Error =>, Status =>)
      Contact( #Flags.Exit_pec_fault )
      S_Coil( #Diag.Alarm[4] )
   END_RUNG
   // the same network as SCL:
   #Program_Alarm[4](SIG := #Diag.Alarm[4], SD_1 := #Device_name, ENO => #_w1);   // Program_Alarm
   IF #_w1 AND #Flags.Exit_pec_fault THEN #Diag.Alarm[4] := TRUE; END_IF;
END_REGION

REGION Network 26: Alarm 5: Encoder fault / Pulssianturin vika
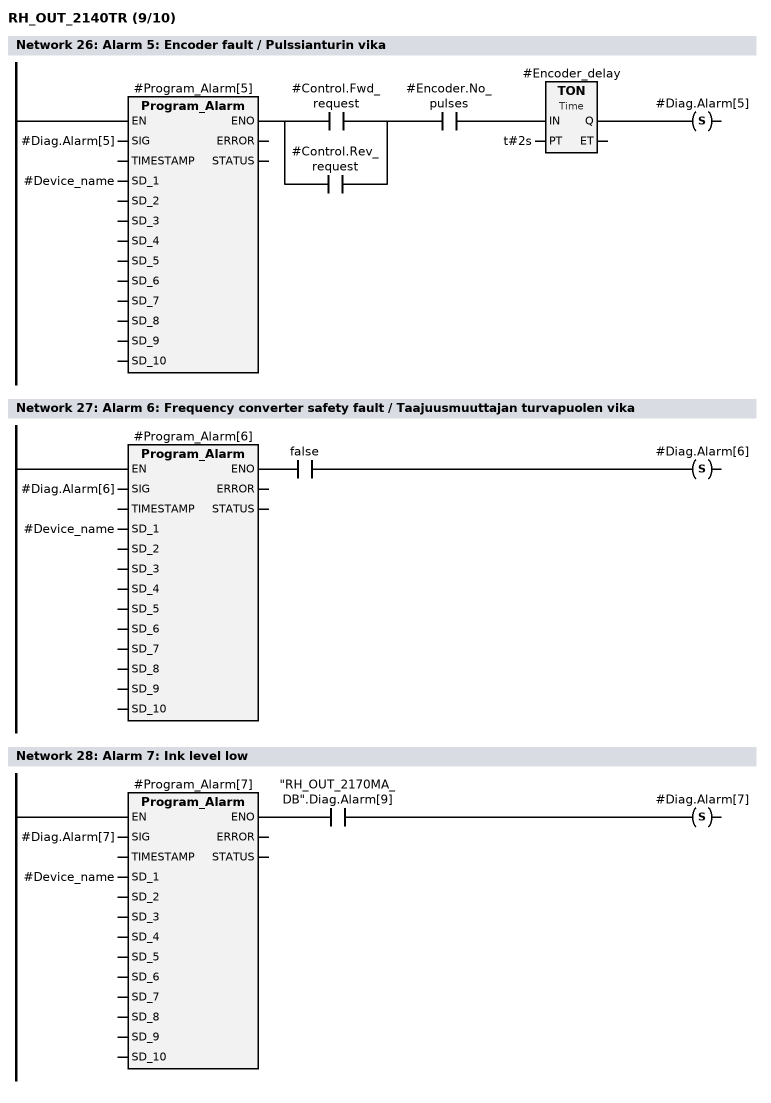
   RUNG wire#powerrail
      #Program_Alarm[5].Program_Alarm(SIG := #Diag.Alarm[5], TIMESTAMP :=, SD_1 := #Device_name, SD_2 :=, SD_3 :=, SD_4 :=, SD_5 :=, SD_6 :=, SD_7 :=, SD_8 :=, SD_9 :=, SD_10 :=, Error =>, Status =>)
      wire#w1
      Contact( #Control.Fwd_request )
      wire#w2
      Contact( #Encoder.No_pulses )
      { S7_Templates := "time_type := Time" } #Encoder_delay.TON(pt := t#2s, et =>)
      S_Coil( #Diag.Alarm[5] )
   END_RUNG
   RUNG wire#w1
      Contact( #Control.Rev_request )
   END_RUNG wire#w2
   // the same network as SCL:
   #Program_Alarm[5](SIG := #Diag.Alarm[5], SD_1 := #Device_name, ENO => #_w1);   // Program_Alarm
   #Encoder_delay(IN := #_w1 AND (#Control.Fwd_request OR #Control.Rev_request) AND #Encoder.No_pulses,   // TON
                  PT := t#2s);
   IF #Encoder_delay.Q THEN #Diag.Alarm[5] := TRUE; END_IF;
END_REGION

REGION Network 27: Alarm 6: Frequency converter safety fault / Taajuusmuuttajan turvapuolen vika
   RUNG wire#powerrail
      #Program_Alarm[6].Program_Alarm(SIG := #Diag.Alarm[6], TIMESTAMP :=, SD_1 := #Device_name, SD_2 :=, SD_3 :=, SD_4 :=, SD_5 :=, SD_6 :=, SD_7 :=, SD_8 :=, SD_9 :=, SD_10 :=, Error =>, Status =>)
      Contact( false )
      S_Coil( #Diag.Alarm[6] )
   END_RUNG
   // the same network as SCL:
   #Program_Alarm[6](SIG := #Diag.Alarm[6], SD_1 := #Device_name, ENO => #_w1);   // Program_Alarm
   IF #_w1 AND false THEN #Diag.Alarm[6] := TRUE; END_IF;
END_REGION

REGION Network 28: Alarm 7: Ink level low
   RUNG wire#powerrail
      #Program_Alarm[7].Program_Alarm(SIG := #Diag.Alarm[7], TIMESTAMP :=, SD_1 := #Device_name, SD_2 :=, SD_3 :=, SD_4 :=, SD_5 :=, SD_6 :=, SD_7 :=, SD_8 :=, SD_9 :=, SD_10 :=, Error =>, Status =>)
      Contact( "RH_OUT_2170MA_DB".Diag.Alarm[9] )
      S_Coil( #Diag.Alarm[7] )
   END_RUNG
   // the same network as SCL:
   #Program_Alarm[7](SIG := #Diag.Alarm[7], SD_1 := #Device_name, ENO => #_w1);   // Program_Alarm
   IF #_w1 AND "RH_OUT_2170MA_DB".Diag.Alarm[9] THEN #Diag.Alarm[7] := TRUE; END_IF;
END_REGION

REGION Network 29: Event 1: Device interlock on / Laitteen lukitus päällä
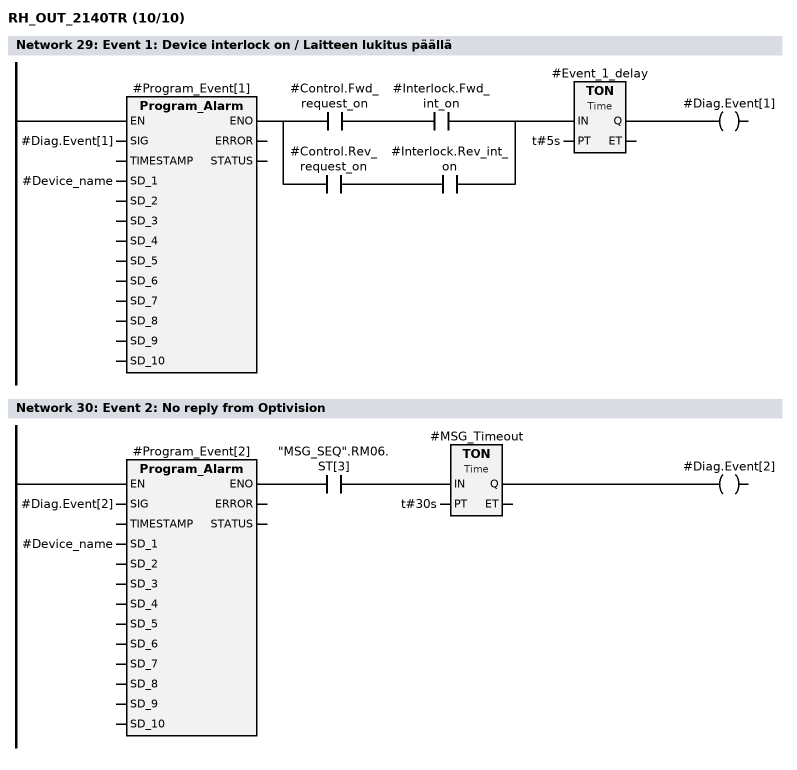
   RUNG wire#powerrail
      #Program_Event[1].Program_Alarm(SIG := #Diag.Event[1], TIMESTAMP :=, SD_1 := #Device_name, SD_2 :=, SD_3 :=, SD_4 :=, SD_5 :=, SD_6 :=, SD_7 :=, SD_8 :=, SD_9 :=, SD_10 :=, Error =>, Status =>)
      wire#w1
      Contact( #Control.Fwd_request_on )
      Contact( #Interlock.Fwd_int_on )
      wire#w2
      { S7_Templates := "time_type := Time" } #Event_1_delay.TON(pt := t#5s, et =>)
      Coil( #Diag.Event[1] )
   END_RUNG
   RUNG wire#w1
      Contact( #Control.Rev_request_on )
      Contact( #Interlock.Rev_int_on )
   END_RUNG wire#w2
   // the same network as SCL:
   #Program_Event[1](SIG := #Diag.Event[1], SD_1 := #Device_name, ENO => #_w1);   // Program_Alarm
   #Event_1_delay(IN := #_w1 AND ((#Control.Fwd_request_on AND #Interlock.Fwd_int_on) OR (#Control.Rev_request_on AND #Interlock.Rev_int_on)),   // TON
                  PT := t#5s);
   #Diag.Event[1] := #Event_1_delay.Q;
END_REGION

REGION Network 30: Event 2: No reply from Optivision
   RUNG wire#powerrail
      #Program_Event[2].Program_Alarm(SIG := #Diag.Event[2], TIMESTAMP :=, SD_1 := #Device_name, SD_2 :=, SD_3 :=, SD_4 :=, SD_5 :=, SD_6 :=, SD_7 :=, SD_8 :=, SD_9 :=, SD_10 :=, Error =>, Status =>)
      Contact( "MSG_SEQ".RM06.ST[3] )
      { S7_Templates := "time_type := Time" } #MSG_Timeout.TON(pt := t#30s, et =>)
      Coil( #Diag.Event[2] )
   END_RUNG
   // the same network as SCL:
   #Program_Event[2](SIG := #Diag.Event[2], SD_1 := #Device_name, ENO => #_w1);   // Program_Alarm
   #MSG_Timeout(IN := #_w1 AND "MSG_SEQ".RM06.ST[3], PT := t#30s);   // TON
   #Diag.Event[2] := #MSG_Timeout.Q;
END_REGION
END_FUNCTION_BLOCK
